FUNCTION_BLOCK ADD_REAL (* IEC 61131-3 REAL Addition *)
  (* Standard: 61131-3 *)
  (* Version 0.1, 2006-09-11, JHC, Holobloc Inc, Converted to Template. *)
  (* Version 0.0, 2004-12-15, JHC, Rockwell Automation, Converted from SRC format. *)
  (* Compiler header: package fb.rt.plc.math; *)
  (* Compiler classdef: ( IN1 + IN2 ) *)
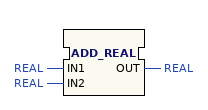
  VAR_INPUT
    IN1 : REAL; (* Augend *)
    IN2 : REAL; (* Addend *)
  END_VAR
  VAR_OUTPUT
    OUT : REAL; (* Sum *)
  END_VAR
END_FUNCTION_BLOCK
